(* PLC project Semaforo.project, CODESYS CODESYS V3.5 SP21 Patch 2 *)
(* stored: creationDateTime 2025-09-16T15:13:17.4947793, modificationDateTime 2025-09-16T14:50:45.2237515 *)

{attribute 'qualified_only'}
{attribute 'strict'}
TYPE Enum_stoplight : (Red, Yellow, Green, Off);
END_TYPE

TYPE Struct_stoplight : STRUCT
  Red : BOOL;
  Yellow : BOOL;
  Green : BOOL;
  Off : BOOL;
END_STRUCT;
END_TYPE

PROGRAM PLC_PRG
  VAR
    Enum_carSL : Enum_stoplight := Enum_stoplight.Green;  (* all stoplight possibile state (Red,Yellow,Green,Off) *)
    Enum_pedSL : Enum_stoplight := Enum_stoplight.Red;  (* same as Enum_carSL but refering to pedestrian stoplight *)
    car_stoplight : Struct_stoplight;  (* stoplight state as BOOL (used in the visu) *)
    ped_stoplight : Struct_stoplight;
    ped_cal : BOOL;  (* TRUE when pedestrian can cross (Green or Yellow)(FALSE when in nightmode) *)
    ped_btn : BOOL;  (* link to request button in visu *)
    night_btn : BOOL;  (* retain button TRUE when in nightmode *)
    night_yellowOn : BOOL;  (* used to "simulate" the pulsing light (nightmode) *)
    TON_carYellowTime : TON;
    car_yellowTime : TIME := TIME#2s0ms;
    TON_pedGreenTime : TON;
    ped_greenTime : TIME := TIME#5s0ms;
    TON_pedYellowTime : TON;
    ped_yellowTime : TIME := TIME#2s0ms;
    TON_yellowLightOn : TON;
    TON_yellowLightOff : TON;
    night_pulsingTime : TIME := TIME#500ms;
  END_VAR
  VAR  (* added by the conversion: wires and edge detectors of the diagram *)
    _w7 : BOOL;
    _w40 : BOOL;
    _w48 : BOOL;
  END_VAR

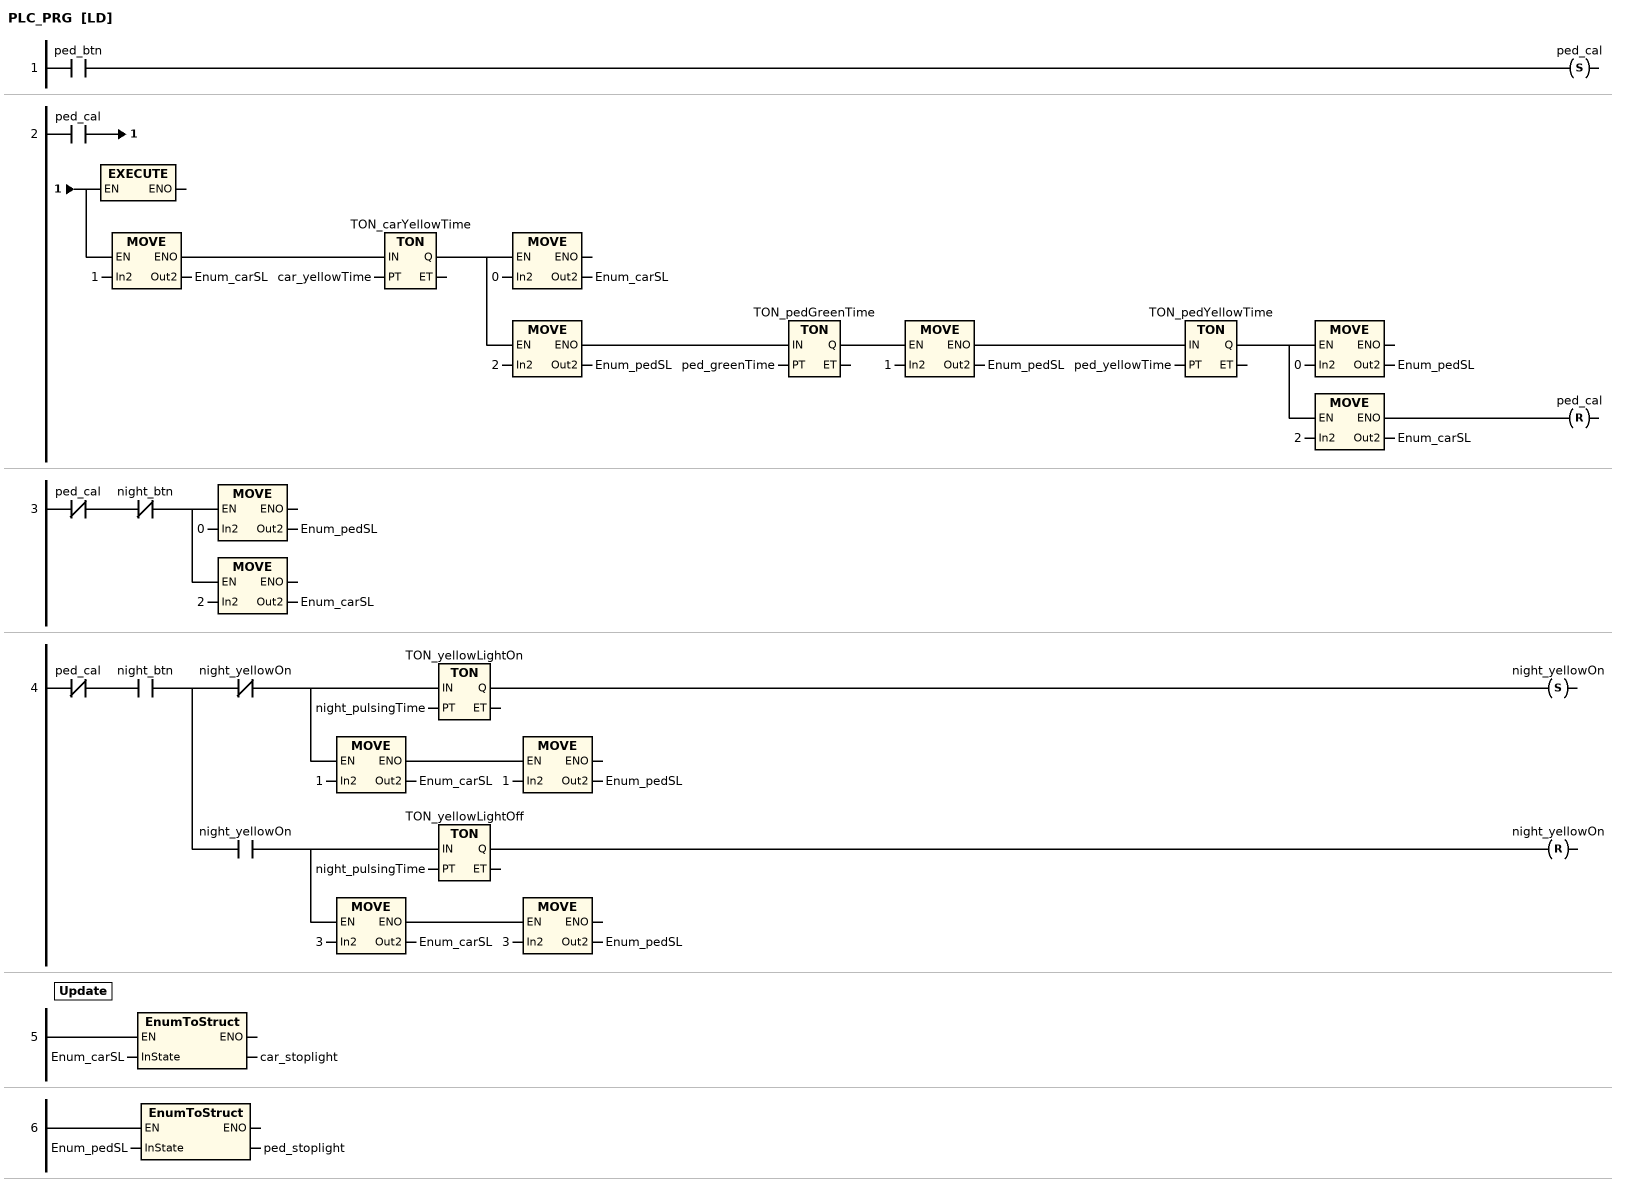
(* LD diagram, written out as Structured Text *)

IF ped_btn THEN ped_cal := TRUE; END_IF;

_w7 := ped_cal;
IF _w7 THEN Enum_carSL := 1; END_IF;
TON_carYellowTime(IN := _w7, PT := car_yellowTime);
IF TON_carYellowTime.Q THEN Enum_carSL := 0; END_IF;
IF TON_carYellowTime.Q THEN Enum_pedSL := 2; END_IF;
TON_pedGreenTime(IN := TON_carYellowTime.Q, PT := ped_greenTime);
IF TON_pedGreenTime.Q THEN Enum_pedSL := 1; END_IF;
TON_pedYellowTime(IN := TON_pedGreenTime.Q, PT := ped_yellowTime);
IF TON_pedYellowTime.Q THEN Enum_carSL := 2; END_IF;
IF TON_pedYellowTime.Q THEN ped_cal := FALSE; END_IF;
IF TON_pedYellowTime.Q THEN Enum_pedSL := 0; END_IF;
IF _w7 THEN
  IF Enum_pedSL = Enum_stoplight.Off THEN
     Enum_pedSL := Enum_stoplight.Yellow;
  END_IF
END_IF;

IF NOT ped_cal AND NOT night_btn THEN Enum_pedSL := 0; END_IF;
IF NOT ped_cal AND NOT night_btn THEN Enum_carSL := 2; END_IF;

_w40 := NOT ped_cal AND night_btn AND NOT night_yellowOn;
TON_yellowLightOn(IN := _w40, PT := night_pulsingTime);
IF TON_yellowLightOn.Q THEN night_yellowOn := TRUE; END_IF;
IF _w40 THEN Enum_carSL := 1; END_IF;
IF _w40 THEN Enum_pedSL := 1; END_IF;
_w48 := NOT ped_cal AND night_btn AND night_yellowOn;
TON_yellowLightOff(IN := _w48, PT := night_pulsingTime);
IF TON_yellowLightOff.Q THEN night_yellowOn := FALSE; END_IF;
IF _w48 THEN Enum_carSL := 3; END_IF;
IF _w48 THEN Enum_pedSL := 3; END_IF;
Update:

car_stoplight := EnumToStruct(InState := Enum_carSL);

ped_stoplight := EnumToStruct(InState := Enum_pedSL);
END_PROGRAM

FUNCTION EnumToStruct : Struct_stoplight
  VAR_INPUT
    InState : Enum_stoplight;
  END_VAR

                    EnumToStruct.Red    := FALSE;
EnumToStruct.Yellow := FALSE;
EnumToStruct.Green  := FALSE;
EnumToStruct.Off    := FALSE;

CASE InState OF
    Enum_stoplight.Red:    EnumToStruct.Red := TRUE;
    Enum_stoplight.Yellow: EnumToStruct.Yellow := TRUE;
    Enum_stoplight.Green:  EnumToStruct.Green := TRUE;
	Enum_stoplight.Off:  EnumToStruct.Off := TRUE;
END_CASE
                  
END_FUNCTION

CONFIGURATION Device
  RESOURCE Application ON PLC
    TASK MainTask(INTERVAL := T#20ms, PRIORITY := 1);
    TASK VISU_TASK(INTERVAL := T#100ms, PRIORITY := 31);
    PROGRAM PLC_PRG WITH MainTask : PLC_PRG;
    PROGRAM VisuElems.Visu_Prg WITH VISU_TASK : VisuElems.Visu_Prg;
  END_RESOURCE
END_CONFIGURATION
